// TIA Portal V16 export
// export: Created 2024-05-10T06:46:41.2862557Z, ExportSetting WithDefaults, DisplayName Totally Integrated Automation Portal, DisplayVersion V16, DisplayName TIA Portal Version Control Interface, DisplayVersion V16, DisplayName TIA Portal Openness, DisplayVersion V16, DisplayName STEP 7 Professional, DisplayVersion V16, DisplayName STEP 7 Safety, DisplayVersion V16, DisplayName WinCC Professional, DisplayVersion V16
FUNCTION_BLOCK "K10_自动"   // FB10, LAD
{ S7_Optimized_Access := 'TRUE' }
VERSION : 0.1
// stored: AutoNumber false, IsIECCheckEnabled false, IsRetainMemResEnabled false, MemoryReserve 100, SetENOAutomatically false, UDAEnableTagReadback false
   VAR_TEMP
      M_OneStep : Bool;   // 单步运行
      M_Pluse : Array[1..10] of Bool;   // 脉冲
      "M_Init Pos1" : Bool;   // 初始位1
      "M_Init Pos2" : Bool;   // 初始位2
   END_VAR
   VAR_TEMP   // added for the SCL form of the ladder/FBD networks
      _w1 : Bool;
   END_VAR
BEGIN

REGION Network 1: 自动条件(立停)
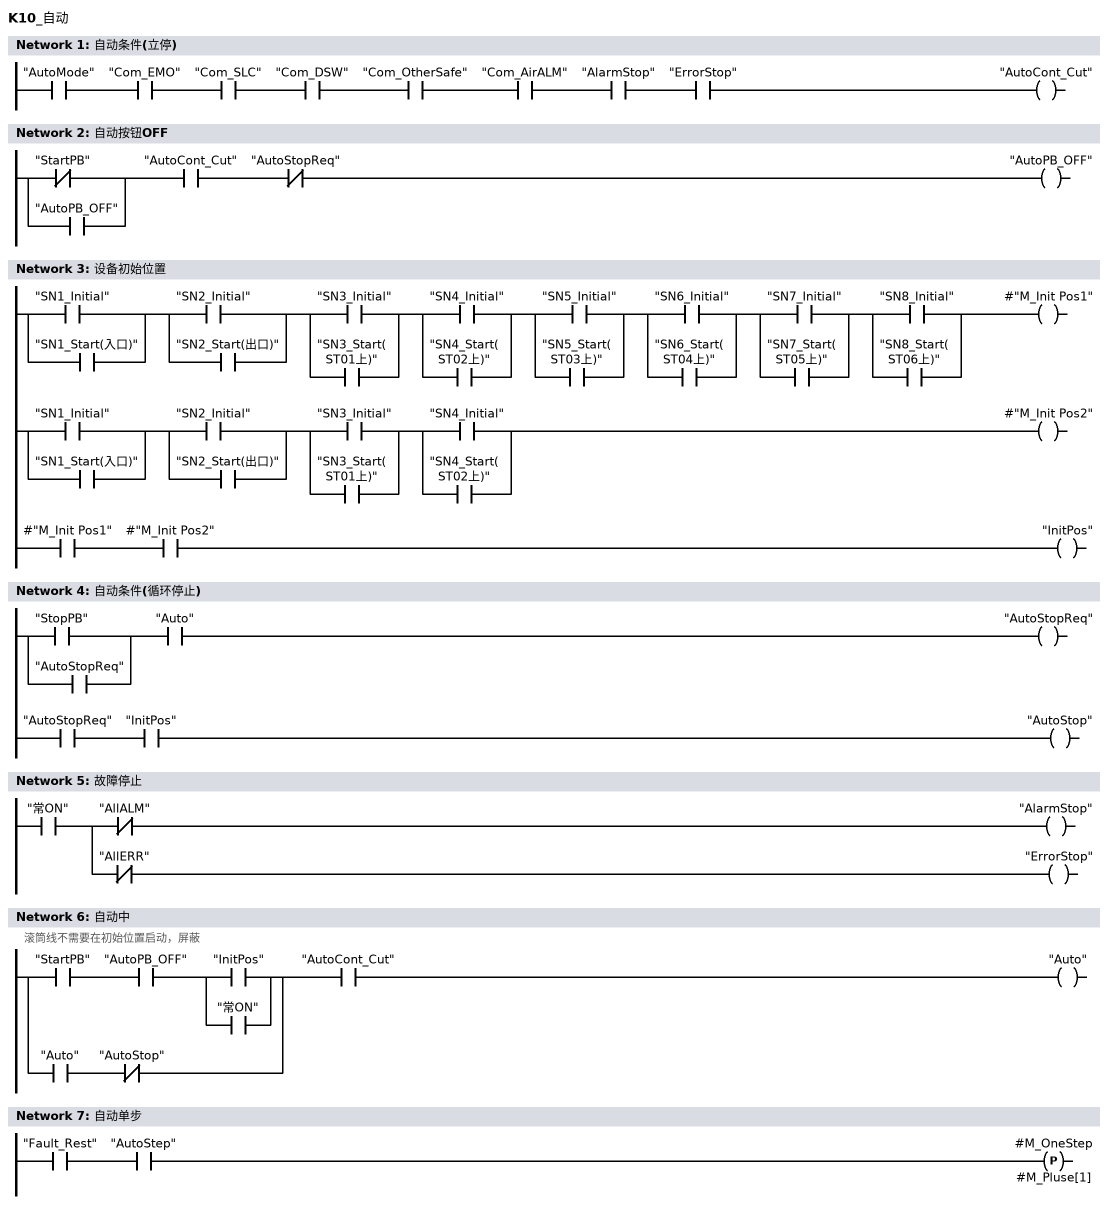
   RUNG wire#powerrail
      Contact( "AutoMode" )
      Contact( "Com_EMO" )
      Contact( "Com_SLC" )
      Contact( "Com_DSW" )
      Contact( "Com_OtherSafe" )
      Contact( "Com_AirALM" )
      Contact( "AlarmStop" )
      Contact( "ErrorStop" )
      Coil( "AutoCont_Cut" )
   END_RUNG
   // the same network as SCL:
   "AutoCont_Cut" := "AutoMode" AND "Com_EMO" AND "Com_SLC" AND "Com_DSW" AND "Com_OtherSafe" AND "Com_AirALM" AND "AlarmStop" AND "ErrorStop";
END_REGION

REGION Network 2: 自动按钮OFF
   RUNG wire#powerrail
      I_Contact( "StartPB" )
      wire#w1
      Contact( "AutoCont_Cut" )
      I_Contact( "AutoStopReq" )
      Coil( "AutoPB_OFF" )
   END_RUNG
   RUNG wire#powerrail
      Contact( "AutoPB_OFF" )
   END_RUNG wire#w1
   // the same network as SCL:
   "AutoPB_OFF" := (NOT "StartPB" OR "AutoPB_OFF") AND "AutoCont_Cut" AND NOT "AutoStopReq";
END_REGION

REGION Network 3: 设备初始位置
   RUNG wire#powerrail
      Contact( "SN1_Initial" )
      wire#w1
      Contact( "SN2_Initial" )
      wire#w2
      Contact( "SN3_Initial" )
      wire#w3
      Contact( "SN4_Initial" )
      wire#w4
      Contact( "SN5_Initial" )
      wire#w5
      Contact( "SN6_Initial" )
      wire#w6
      Contact( "SN7_Initial" )
      wire#w7
      Contact( "SN8_Initial" )
      wire#w8
      Coil( #"M_Init Pos1" )
   END_RUNG
   RUNG wire#powerrail
      Contact( "SN1_Start(入口)" )
   END_RUNG wire#w1
   RUNG wire#w1
      Contact( "SN2_Start(出口)" )
   END_RUNG wire#w2
   RUNG wire#w2
      Contact( "SN3_Start(ST01上)" )
   END_RUNG wire#w3
   RUNG wire#w3
      Contact( "SN4_Start(ST02上)" )
   END_RUNG wire#w4
   RUNG wire#w4
      Contact( "SN5_Start(ST03上)" )
   END_RUNG wire#w5
   RUNG wire#w5
      Contact( "SN6_Start(ST04上)" )
   END_RUNG wire#w6
   RUNG wire#w6
      Contact( "SN7_Start(ST05上)" )
   END_RUNG wire#w7
   RUNG wire#w7
      Contact( "SN8_Start(ST06上)" )
   END_RUNG wire#w8
   RUNG wire#powerrail
      Contact( "SN1_Initial" )
      wire#w9
      Contact( "SN2_Initial" )
      wire#w10
      Contact( "SN3_Initial" )
      wire#w11
      Contact( "SN4_Initial" )
      wire#w12
      Coil( #"M_Init Pos2" )
   END_RUNG
   RUNG wire#powerrail
      Contact( "SN1_Start(入口)" )
   END_RUNG wire#w9
   RUNG wire#w9
      Contact( "SN2_Start(出口)" )
   END_RUNG wire#w10
   RUNG wire#w10
      Contact( "SN3_Start(ST01上)" )
   END_RUNG wire#w11
   RUNG wire#w11
      Contact( "SN4_Start(ST02上)" )
   END_RUNG wire#w12
   RUNG wire#powerrail
      Contact( #"M_Init Pos1" )
      Contact( #"M_Init Pos2" )
      Coil( "InitPos" )
   END_RUNG
   // the same network as SCL:
   #"M_Init Pos1" := ("SN1_Initial" OR "SN1_Start(入口)") AND ("SN2_Initial" OR "SN2_Start(出口)") AND ("SN3_Initial" OR "SN3_Start(ST01上)") AND ("SN4_Initial" OR "SN4_Start(ST02上)") AND ("SN5_Initial" OR "SN5_Start(ST03上)") AND ("SN6_Initial" OR "SN6_Start(ST04上)") AND ("SN7_Initial" OR "SN7_Start(ST05上)") AND ("SN8_Initial" OR "SN8_Start(ST06上)");
   #"M_Init Pos2" := ("SN1_Initial" OR "SN1_Start(入口)") AND ("SN2_Initial" OR "SN2_Start(出口)") AND ("SN3_Initial" OR "SN3_Start(ST01上)") AND ("SN4_Initial" OR "SN4_Start(ST02上)");
   "InitPos" := #"M_Init Pos1" AND #"M_Init Pos2";
END_REGION

REGION Network 4: 自动条件(循环停止)
   RUNG wire#powerrail
      Contact( "StopPB" )
      wire#w1
      Contact( "Auto" )
      Coil( "AutoStopReq" )
   END_RUNG
   RUNG wire#powerrail
      Contact( "AutoStopReq" )
   END_RUNG wire#w1
   RUNG wire#powerrail
      Contact( "AutoStopReq" )
      Contact( "InitPos" )
      Coil( "AutoStop" )
   END_RUNG
   // the same network as SCL:
   "AutoStopReq" := ("StopPB" OR "AutoStopReq") AND "Auto";
   "AutoStop" := "AutoStopReq" AND "InitPos";
END_REGION

REGION Network 5: 故障停止
   RUNG wire#powerrail
      Contact( "常ON" )
      wire#w1
      I_Contact( "AllALM" )
      Coil( "AlarmStop" )
   END_RUNG
   RUNG wire#w1
      I_Contact( "AllERR" )
      Coil( "ErrorStop" )
   END_RUNG
   // the same network as SCL:
   "AlarmStop" := "常ON" AND NOT "AllALM";
   "ErrorStop" := "常ON" AND NOT "AllERR";
END_REGION

REGION Network 6: 自动中
   // 滚筒线不需要在初始位置启动，屏蔽
   RUNG wire#powerrail
      Contact( "StartPB" )
      Contact( "AutoPB_OFF" )
      wire#w1
      Contact( "InitPos" )
      wire#w2
      Contact( "AutoCont_Cut" )
      Coil( "Auto" )
   END_RUNG
   RUNG wire#w1
      Contact( "常ON" )
   END_RUNG wire#w2
   RUNG wire#powerrail
      Contact( "Auto" )
      I_Contact( "AutoStop" )
   END_RUNG wire#w2
   // the same network as SCL:
   "Auto" := (("StartPB" AND "AutoPB_OFF" AND ("InitPos" OR "常ON")) OR ("Auto" AND NOT "AutoStop")) AND "AutoCont_Cut";
END_REGION

REGION Network 7: 自动单步
   #_w1 := "Fault_Rest" AND "AutoStep";
   #M_OneStep := #_w1 AND NOT #M_Pluse[1];   // rising edge
   #M_Pluse[1] := #_w1;
END_REGION
END_FUNCTION_BLOCK
